// TIA Portal V20 export
FUNCTION "LIT100" : Void   // FC6, FBD
{ S7_Optimized_Access := 'TRUE' }
// stored: SetENOAutomatically false
BEGIN

REGION Network 1: Channel input
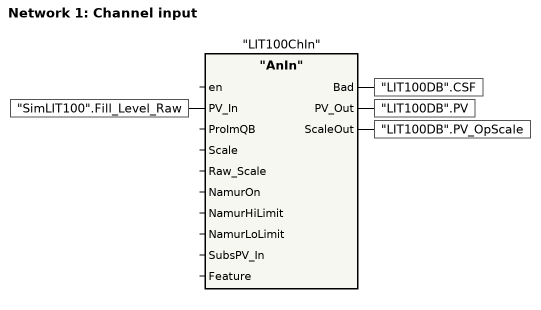
   "LIT100ChIn"(PV_In := "SimLIT100".Fill_Level_Raw,   // "AnIn"
                Bad => "LIT100DB".CSF,
                PV_Out => "LIT100DB".PV,
                ScaleOut => "LIT100DB".PV_OpScale);
END_REGION

REGION Network 2: PIDConL
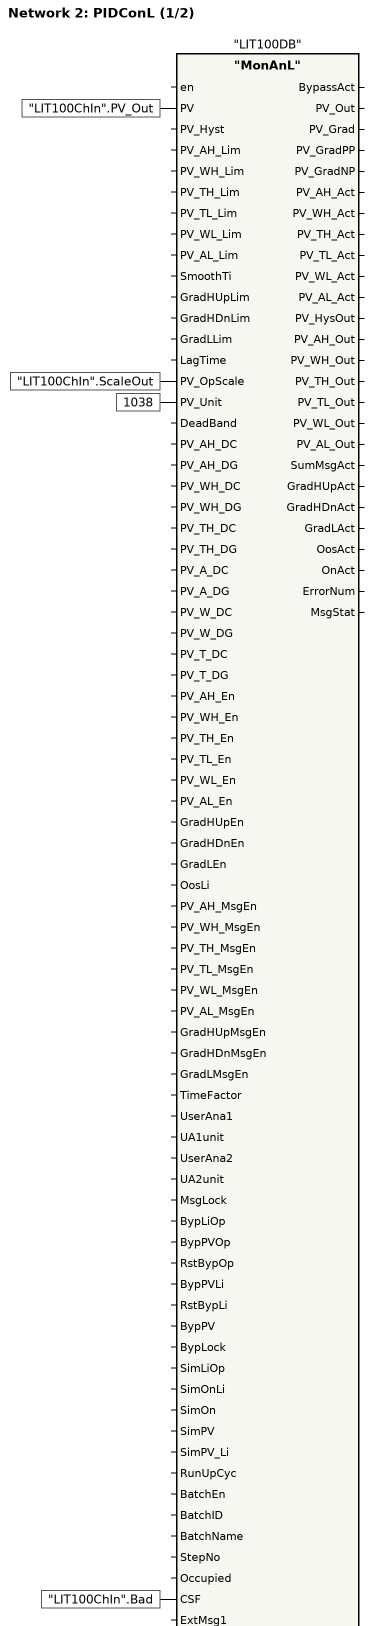
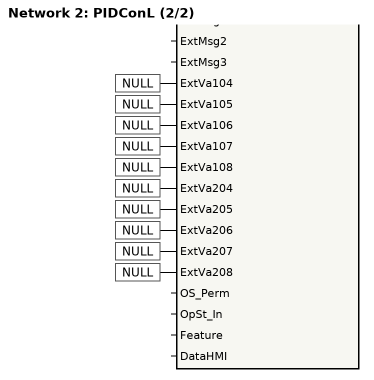
   "LIT100DB"(PV := "LIT100ChIn".PV_Out,   // "MonAnL"
              PV_OpScale := "LIT100ChIn".ScaleOut,
              PV_Unit := 1038,
              CSF := "LIT100ChIn".Bad,
              ExtVa104 := NULL,
              ExtVa105 := NULL,
              ExtVa106 := NULL,
              ExtVa107 := NULL,
              ExtVa108 := NULL,
              ExtVa204 := NULL,
              ExtVa205 := NULL,
              ExtVa206 := NULL,
              ExtVa207 := NULL,
              ExtVa208 := NULL);
END_REGION

REGION Network 3: MTP
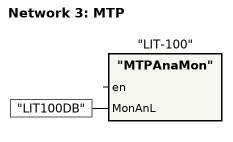
   "LIT-100"(MonAnL := "LIT100DB");   // "MTPAnaMon"
END_REGION
END_FUNCTION
